% RSLogix 500 project Project - Five_Conveyor_System.RSS, saved by version 8.30.00.16 %
PROJECT "UNTITLED"    % processor: Bul.1763 MicroLogix 1100 Series B %

PROGRAM FILES
  LAD 2 "MAIN"  8 rungs
  LAD 3 "BELT 1"  8 rungs  % Conveyor 1 %
  LAD 4 "BELT 2"  8 rungs  % CONVEYOR 2 %
  LAD 5 "BELT 3"  8 rungs  % CONVEYOR 3 %
  LAD 6 "BELT 4"  8 rungs  % CONVEYOR 4 %
  LAD 7 "BELT 5"  8 rungs  % CONVEYOR 5 %
  LAD 8 "SEQUENCE"  14 rungs  % CONVEYOR OPERATION %

DATA FILES
  O0 OUTPUT  4 elements
  I1 INPUT  6 elements
  S2 STATUS  66 elements
  B3 BINARY  5 elements
  T4 TIMER  25 elements
  C5 COUNTER  5 elements
  R6 CONTROL  1 elements
  N7 INTEGER  5 elements
  F8 FLOAT  1 elements

LADDER 2 "MAIN"
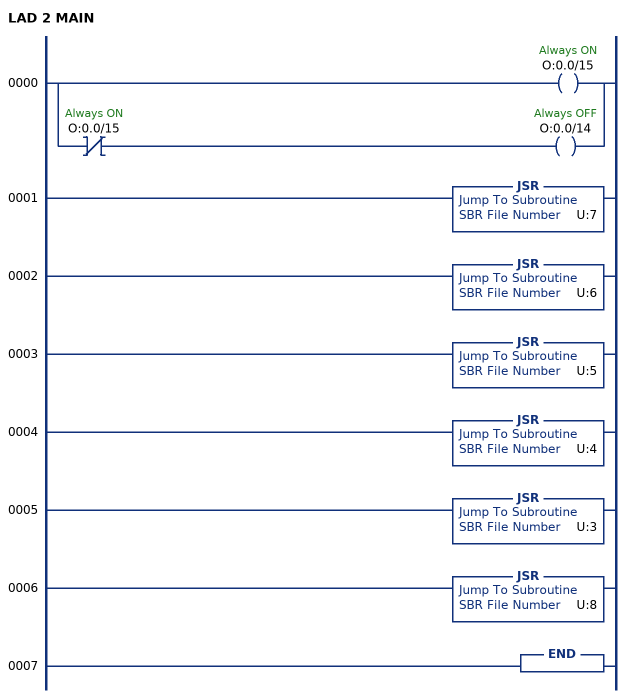
% Rung: 0 %
SOR BST OTE O:0.0/15 NXB XIO O:0.0/15 OTE O:0.0/14 BND EOR
%   O:0.0/15  "Always ON" %
%   O:0.0/14  "Always OFF" %
% Rung: 1 %
SOR JSR U:7 EOR
% Rung: 2 %
SOR JSR U:6 EOR
% Rung: 3 %
SOR JSR U:5 EOR
% Rung: 4 %
SOR JSR U:4 EOR
% Rung: 5 %
SOR JSR U:3 EOR
% Rung: 6 %
SOR JSR U:8 EOR
% Rung: 7 %
SOR END EOR

LADDER 3 "BELT 1"    % Conveyor 1 %
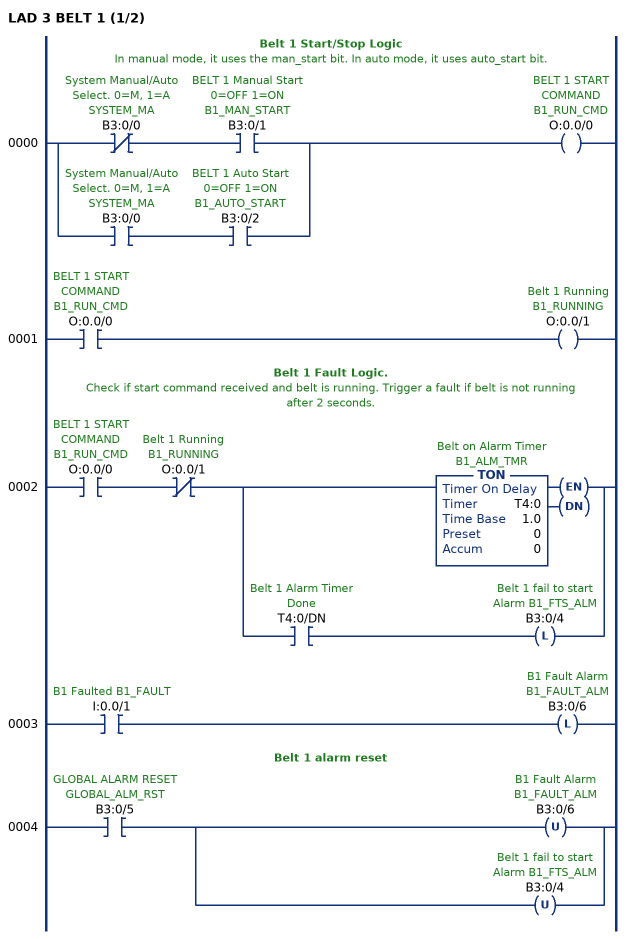
% Rung: 0 %
% TITLE: Belt 1 Start/Stop Logic %
% In manual mode, it uses the man_start bit. In auto mode, it uses auto_start bit. %
SOR BST XIO B3:0/0 XIC B3:0/1 NXB XIC B3:0/0 XIC B3:0/2 BND OTE O:0.0/0 EOR
%   B3:0/0  SYSTEM_MA  "System Manual/Auto Select. 0=M, 1=A" %
%   B3:0/1  B1_MAN_START  "BELT 1 Manual Start 0=OFF 1=ON" %
%   B3:0/2  B1_AUTO_START  "BELT 1 Auto Start 0=OFF 1=ON" %
%   O:0.0/0  B1_RUN_CMD  "BELT 1 START COMMAND" %
% Rung: 1 %
SOR XIC O:0.0/0 OTE O:0.0/1 EOR
%   O:0.0/0  B1_RUN_CMD  "BELT 1 START COMMAND" %
%   O:0.0/1  B1_RUNNING  "Belt 1 Running" %
% Rung: 2 %
% TITLE: Belt 1 Fault Logic. %
% Check if start command received and belt is running. Trigger a fault if belt is not running after 2 seconds. %
SOR XIC O:0.0/0 XIO O:0.0/1 BST TON T4:0 1.0 0 0 NXB XIC T4:0/DN OTL B3:0/4 BND EOR
%   O:0.0/0  B1_RUN_CMD  "BELT 1 START COMMAND" %
%   O:0.0/1  B1_RUNNING  "Belt 1 Running" %
%   T4:0  B1_ALM_TMR  "Belt on Alarm Timer" %
%   T4:0/DN  "Belt 1 Alarm Timer Done" %
%   B3:0/4  B1_FTS_ALM  "Belt 1 fail to start Alarm" %
% Rung: 3 %
SOR XIC I:0.0/1 OTL B3:0/6 EOR
%   I:0.0/1  B1_FAULT  "B1 Faulted" %
%   B3:0/6  B1_FAULT_ALM  "B1 Fault Alarm" %
% Rung: 4 %
% TITLE: Belt 1 alarm reset %
SOR XIC B3:0/5 BST OTU B3:0/6 NXB OTU B3:0/4 BND EOR
%   B3:0/5  GLOBAL_ALM_RST  "GLOBAL ALARM RESET" %
%   B3:0/6  B1_FAULT_ALM  "B1 Fault Alarm" %
%   B3:0/4  B1_FTS_ALM  "Belt 1 fail to start Alarm" %

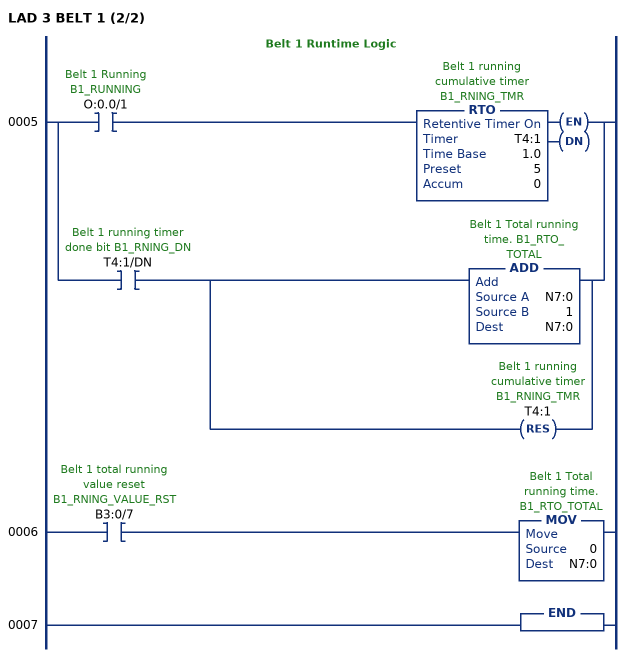
% Rung: 5 %
% TITLE: Belt 1 Runtime Logic %
SOR BST XIC O:0.0/1 RTO T4:1 1.0 5 0 NXB XIC T4:1/DN BST ADD N7:0 1 N7:0 NXB RES T4:1 BND BND EOR
%   O:0.0/1  B1_RUNNING  "Belt 1 Running" %
%   T4:1  B1_RNING_TMR  "Belt 1 running cumulative timer" %
%   T4:1/DN  B1_RNING_DN  "Belt 1 running timer done bit" %
%   N7:0  B1_RTO_TOTAL  "Belt 1 Total running time." %
% Rung: 6 %
SOR XIC B3:0/7 MOV 0 N7:0 EOR
%   B3:0/7  B1_RNING_VALUE_RST  "Belt 1 total running value reset" %
%   N7:0  B1_RTO_TOTAL  "Belt 1 Total running time." %
% Rung: 7 %
SOR END EOR

LADDER 4 "BELT 2"    % CONVEYOR 2 %
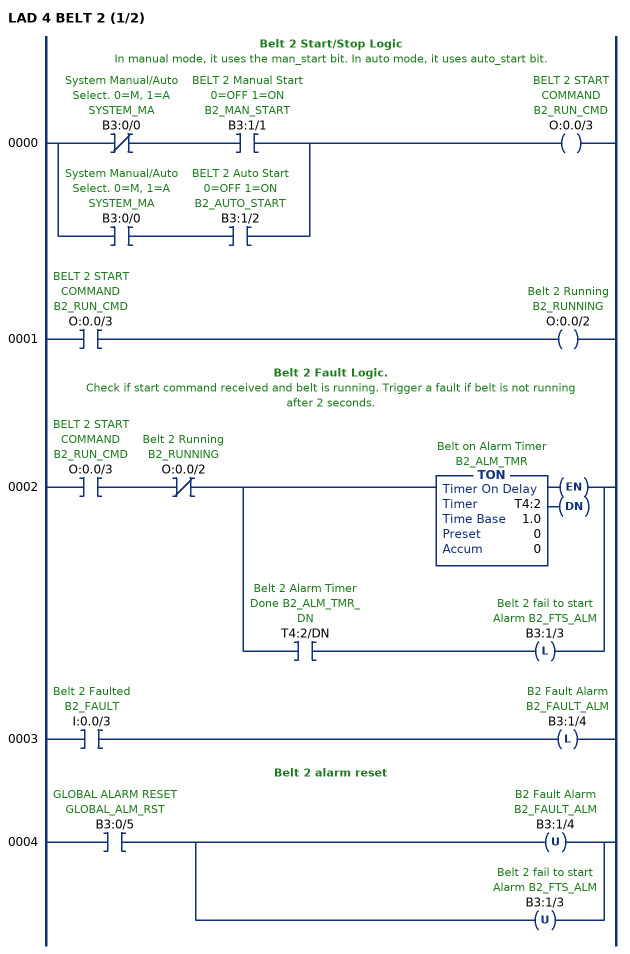
% Rung: 0 %
% TITLE: Belt 2 Start/Stop Logic %
% In manual mode, it uses the man_start bit. In auto mode, it uses auto_start bit. %
SOR BST XIO B3:0/0 XIC B3:1/1 NXB XIC B3:0/0 XIC B3:1/2 BND OTE O:0.0/3 EOR
%   B3:0/0  SYSTEM_MA  "System Manual/Auto Select. 0=M, 1=A" %
%   B3:1/1  B2_MAN_START  "BELT 2 Manual Start 0=OFF 1=ON" %
%   B3:1/2  B2_AUTO_START  "BELT 2 Auto Start 0=OFF 1=ON" %
%   O:0.0/3  B2_RUN_CMD  "BELT 2 START COMMAND" %
% Rung: 1 %
SOR XIC O:0.0/3 OTE O:0.0/2 EOR
%   O:0.0/3  B2_RUN_CMD  "BELT 2 START COMMAND" %
%   O:0.0/2  B2_RUNNING  "Belt 2 Running" %
% Rung: 2 %
% TITLE: Belt 2 Fault Logic. %
% Check if start command received and belt is running. Trigger a fault if belt is not running after 2 seconds. %
SOR XIC O:0.0/3 XIO O:0.0/2 BST TON T4:2 1.0 0 0 NXB XIC T4:2/DN OTL B3:1/3 BND EOR
%   O:0.0/3  B2_RUN_CMD  "BELT 2 START COMMAND" %
%   O:0.0/2  B2_RUNNING  "Belt 2 Running" %
%   T4:2  B2_ALM_TMR  "Belt on Alarm Timer" %
%   T4:2/DN  B2_ALM_TMR_DN  "Belt 2 Alarm Timer Done" %
%   B3:1/3  B2_FTS_ALM  "Belt 2 fail to start Alarm" %
% Rung: 3 %
SOR XIC I:0.0/3 OTL B3:1/4 EOR
%   I:0.0/3  B2_FAULT  "Belt 2 Faulted" %
%   B3:1/4  B2_FAULT_ALM  "B2 Fault Alarm" %
% Rung: 4 %
% TITLE: Belt 2 alarm reset %
SOR XIC B3:0/5 BST OTU B3:1/4 NXB OTU B3:1/3 BND EOR
%   B3:0/5  GLOBAL_ALM_RST  "GLOBAL ALARM RESET" %
%   B3:1/4  B2_FAULT_ALM  "B2 Fault Alarm" %
%   B3:1/3  B2_FTS_ALM  "Belt 2 fail to start Alarm" %

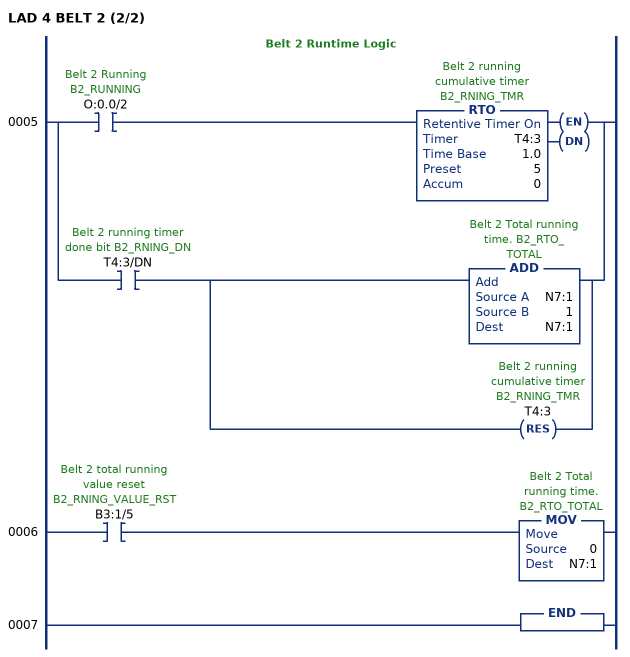
% Rung: 5 %
% TITLE: Belt 2 Runtime Logic %
SOR BST XIC O:0.0/2 RTO T4:3 1.0 5 0 NXB XIC T4:3/DN BST ADD N7:1 1 N7:1 NXB RES T4:3 BND BND EOR
%   O:0.0/2  B2_RUNNING  "Belt 2 Running" %
%   T4:3  B2_RNING_TMR  "Belt 2 running cumulative timer" %
%   T4:3/DN  B2_RNING_DN  "Belt 2 running timer done bit" %
%   N7:1  B2_RTO_TOTAL  "Belt 2 Total running time." %
% Rung: 6 %
SOR XIC B3:1/5 MOV 0 N7:1 EOR
%   B3:1/5  B2_RNING_VALUE_RST  "Belt 2 total running value reset" %
%   N7:1  B2_RTO_TOTAL  "Belt 2 Total running time." %
% Rung: 7 %
SOR END EOR

LADDER 5 "BELT 3"    % CONVEYOR 3 %
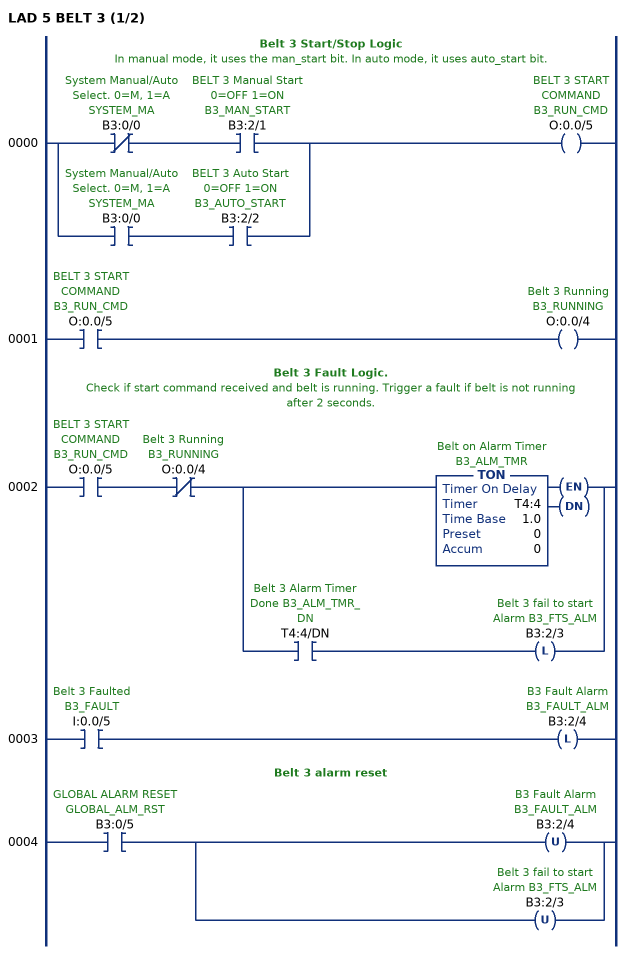
% Rung: 0 %
% TITLE: Belt 3 Start/Stop Logic %
% In manual mode, it uses the man_start bit. In auto mode, it uses auto_start bit. %
SOR BST XIO B3:0/0 XIC B3:2/1 NXB XIC B3:0/0 XIC B3:2/2 BND OTE O:0.0/5 EOR
%   B3:0/0  SYSTEM_MA  "System Manual/Auto Select. 0=M, 1=A" %
%   B3:2/1  B3_MAN_START  "BELT 3 Manual Start 0=OFF 1=ON" %
%   B3:2/2  B3_AUTO_START  "BELT 3 Auto Start 0=OFF 1=ON" %
%   O:0.0/5  B3_RUN_CMD  "BELT 3 START COMMAND" %
% Rung: 1 %
SOR XIC O:0.0/5 OTE O:0.0/4 EOR
%   O:0.0/5  B3_RUN_CMD  "BELT 3 START COMMAND" %
%   O:0.0/4  B3_RUNNING  "Belt 3 Running" %
% Rung: 2 %
% TITLE: Belt 3 Fault Logic. %
% Check if start command received and belt is running. Trigger a fault if belt is not running after 2 seconds. %
SOR XIC O:0.0/5 XIO O:0.0/4 BST TON T4:4 1.0 0 0 NXB XIC T4:4/DN OTL B3:2/3 BND EOR
%   O:0.0/5  B3_RUN_CMD  "BELT 3 START COMMAND" %
%   O:0.0/4  B3_RUNNING  "Belt 3 Running" %
%   T4:4  B3_ALM_TMR  "Belt on Alarm Timer" %
%   T4:4/DN  B3_ALM_TMR_DN  "Belt 3 Alarm Timer Done" %
%   B3:2/3  B3_FTS_ALM  "Belt 3 fail to start Alarm" %
% Rung: 3 %
SOR XIC I:0.0/5 OTL B3:2/4 EOR
%   I:0.0/5  B3_FAULT  "Belt 3 Faulted" %
%   B3:2/4  B3_FAULT_ALM  "B3 Fault Alarm" %
% Rung: 4 %
% TITLE: Belt 3 alarm reset %
SOR XIC B3:0/5 BST OTU B3:2/4 NXB OTU B3:2/3 BND EOR
%   B3:0/5  GLOBAL_ALM_RST  "GLOBAL ALARM RESET" %
%   B3:2/4  B3_FAULT_ALM  "B3 Fault Alarm" %
%   B3:2/3  B3_FTS_ALM  "Belt 3 fail to start Alarm" %

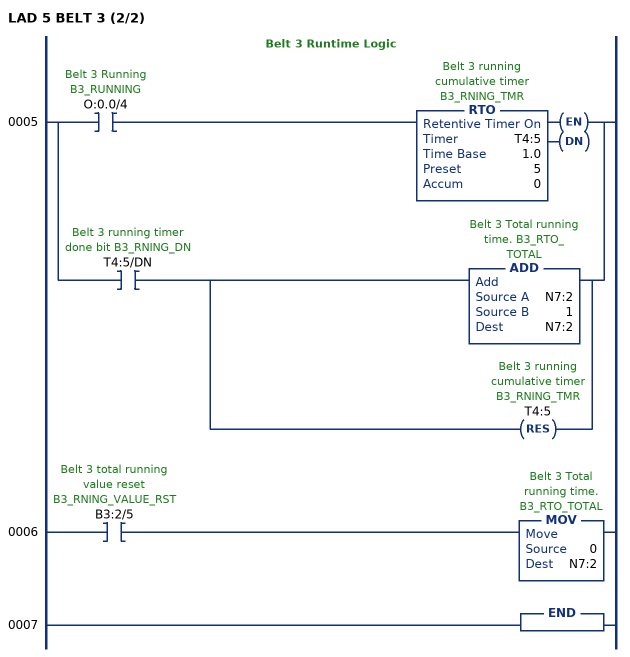
% Rung: 5 %
% TITLE: Belt 3 Runtime Logic %
SOR BST XIC O:0.0/4 RTO T4:5 1.0 5 0 NXB XIC T4:5/DN BST ADD N7:2 1 N7:2 NXB RES T4:5 BND BND EOR
%   O:0.0/4  B3_RUNNING  "Belt 3 Running" %
%   T4:5  B3_RNING_TMR  "Belt 3 running cumulative timer" %
%   T4:5/DN  B3_RNING_DN  "Belt 3 running timer done bit" %
%   N7:2  B3_RTO_TOTAL  "Belt 3 Total running time." %
% Rung: 6 %
SOR XIC B3:2/5 MOV 0 N7:2 EOR
%   B3:2/5  B3_RNING_VALUE_RST  "Belt 3 total running value reset" %
%   N7:2  B3_RTO_TOTAL  "Belt 3 Total running time." %
% Rung: 7 %
SOR END EOR

LADDER 6 "BELT 4"    % CONVEYOR 4 %
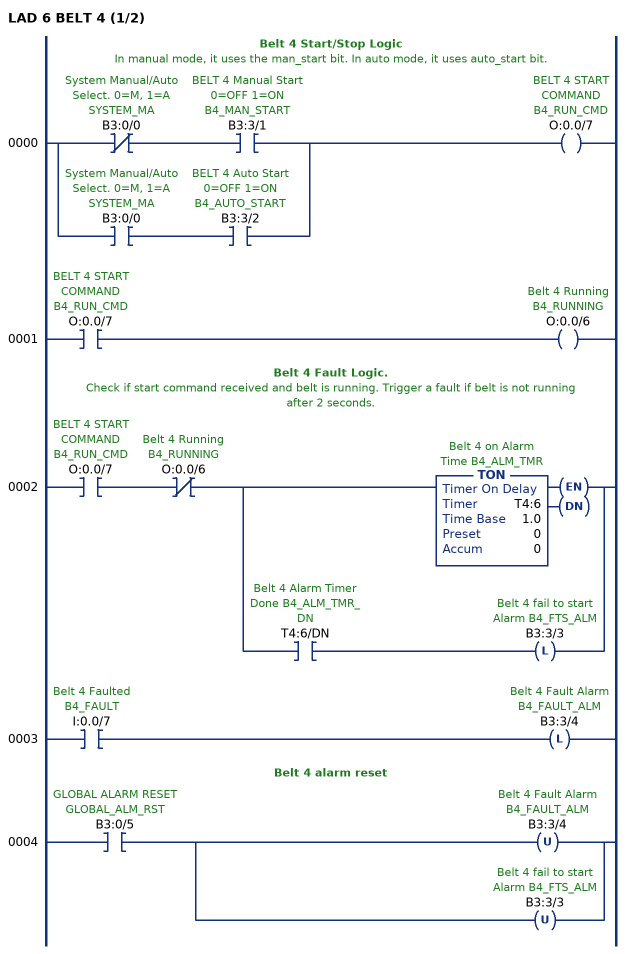
% Rung: 0 %
% TITLE: Belt 4 Start/Stop Logic %
% In manual mode, it uses the man_start bit. In auto mode, it uses auto_start bit. %
SOR BST XIO B3:0/0 XIC B3:3/1 NXB XIC B3:0/0 XIC B3:3/2 BND OTE O:0.0/7 EOR
%   B3:0/0  SYSTEM_MA  "System Manual/Auto Select. 0=M, 1=A" %
%   B3:3/1  B4_MAN_START  "BELT 4 Manual Start 0=OFF 1=ON" %
%   B3:3/2  B4_AUTO_START  "BELT 4 Auto Start 0=OFF 1=ON" %
%   O:0.0/7  B4_RUN_CMD  "BELT 4 START COMMAND" %
% Rung: 1 %
SOR XIC O:0.0/7 OTE O:0.0/6 EOR
%   O:0.0/7  B4_RUN_CMD  "BELT 4 START COMMAND" %
%   O:0.0/6  B4_RUNNING  "Belt 4 Running" %
% Rung: 2 %
% TITLE: Belt 4 Fault Logic. %
% Check if start command received and belt is running. Trigger a fault if belt is not running after 2 seconds. %
SOR XIC O:0.0/7 XIO O:0.0/6 BST TON T4:6 1.0 0 0 NXB XIC T4:6/DN OTL B3:3/3 BND EOR
%   O:0.0/7  B4_RUN_CMD  "BELT 4 START COMMAND" %
%   O:0.0/6  B4_RUNNING  "Belt 4 Running" %
%   T4:6  B4_ALM_TMR  "Belt 4 on Alarm Time" %
%   T4:6/DN  B4_ALM_TMR_DN  "Belt 4 Alarm Timer Done" %
%   B3:3/3  B4_FTS_ALM  "Belt 4 fail to start Alarm" %
% Rung: 3 %
SOR XIC I:0.0/7 OTL B3:3/4 EOR
%   I:0.0/7  B4_FAULT  "Belt 4 Faulted" %
%   B3:3/4  B4_FAULT_ALM  "Belt 4 Fault Alarm" %
% Rung: 4 %
% TITLE: Belt 4 alarm reset %
SOR XIC B3:0/5 BST OTU B3:3/4 NXB OTU B3:3/3 BND EOR
%   B3:0/5  GLOBAL_ALM_RST  "GLOBAL ALARM RESET" %
%   B3:3/4  B4_FAULT_ALM  "Belt 4 Fault Alarm" %
%   B3:3/3  B4_FTS_ALM  "Belt 4 fail to start Alarm" %

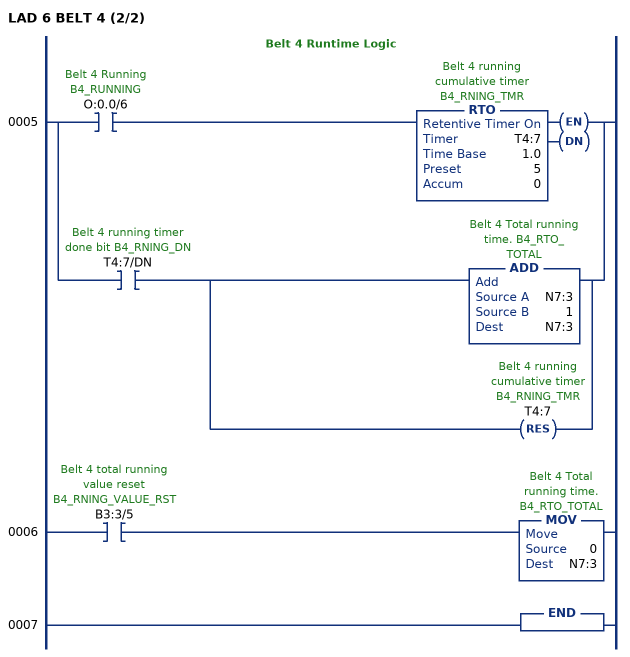
% Rung: 5 %
% TITLE: Belt 4 Runtime Logic %
SOR BST XIC O:0.0/6 RTO T4:7 1.0 5 0 NXB XIC T4:7/DN BST ADD N7:3 1 N7:3 NXB RES T4:7 BND BND EOR
%   O:0.0/6  B4_RUNNING  "Belt 4 Running" %
%   T4:7  B4_RNING_TMR  "Belt 4 running cumulative timer" %
%   T4:7/DN  B4_RNING_DN  "Belt 4 running timer done bit" %
%   N7:3  B4_RTO_TOTAL  "Belt 4 Total running time." %
% Rung: 6 %
SOR XIC B3:3/5 MOV 0 N7:3 EOR
%   B3:3/5  B4_RNING_VALUE_RST  "Belt 4 total running value reset" %
%   N7:3  B4_RTO_TOTAL  "Belt 4 Total running time." %
% Rung: 7 %
SOR END EOR

LADDER 7 "BELT 5"    % CONVEYOR 5 %
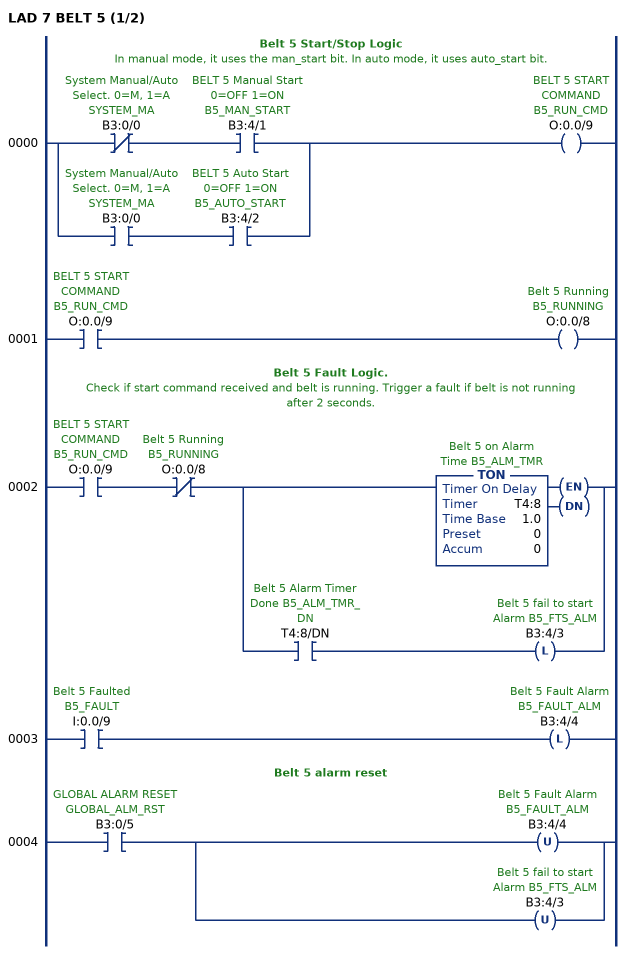
% Rung: 0 %
% TITLE: Belt 5 Start/Stop Logic %
% In manual mode, it uses the man_start bit. In auto mode, it uses auto_start bit. %
SOR BST XIO B3:0/0 XIC B3:4/1 NXB XIC B3:0/0 XIC B3:4/2 BND OTE O:0.0/9 EOR
%   B3:0/0  SYSTEM_MA  "System Manual/Auto Select. 0=M, 1=A" %
%   B3:4/1  B5_MAN_START  "BELT 5 Manual Start 0=OFF 1=ON" %
%   B3:4/2  B5_AUTO_START  "BELT 5 Auto Start 0=OFF 1=ON" %
%   O:0.0/9  B5_RUN_CMD  "BELT 5 START COMMAND" %
% Rung: 1 %
SOR XIC O:0.0/9 OTE O:0.0/8 EOR
%   O:0.0/9  B5_RUN_CMD  "BELT 5 START COMMAND" %
%   O:0.0/8  B5_RUNNING  "Belt 5 Running" %
% Rung: 2 %
% TITLE: Belt 5 Fault Logic. %
% Check if start command received and belt is running. Trigger a fault if belt is not running after 2 seconds. %
SOR XIC O:0.0/9 XIO O:0.0/8 BST TON T4:8 1.0 0 0 NXB XIC T4:8/DN OTL B3:4/3 BND EOR
%   O:0.0/9  B5_RUN_CMD  "BELT 5 START COMMAND" %
%   O:0.0/8  B5_RUNNING  "Belt 5 Running" %
%   T4:8  B5_ALM_TMR  "Belt 5 on Alarm Time" %
%   T4:8/DN  B5_ALM_TMR_DN  "Belt 5 Alarm Timer Done" %
%   B3:4/3  B5_FTS_ALM  "Belt 5 fail to start Alarm" %
% Rung: 3 %
SOR XIC I:0.0/9 OTL B3:4/4 EOR
%   I:0.0/9  B5_FAULT  "Belt 5 Faulted" %
%   B3:4/4  B5_FAULT_ALM  "Belt 5 Fault Alarm" %
% Rung: 4 %
% TITLE: Belt 5 alarm reset %
SOR XIC B3:0/5 BST OTU B3:4/4 NXB OTU B3:4/3 BND EOR
%   B3:0/5  GLOBAL_ALM_RST  "GLOBAL ALARM RESET" %
%   B3:4/4  B5_FAULT_ALM  "Belt 5 Fault Alarm" %
%   B3:4/3  B5_FTS_ALM  "Belt 5 fail to start Alarm" %

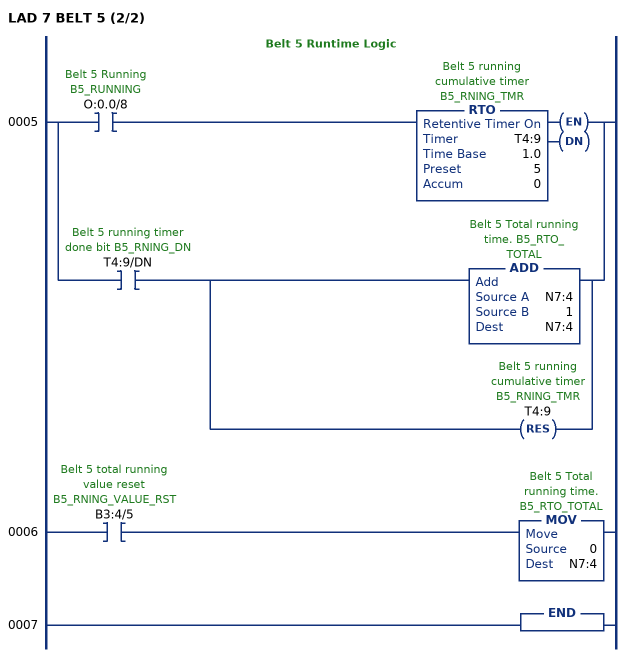
% Rung: 5 %
% TITLE: Belt 5 Runtime Logic %
SOR BST XIC O:0.0/8 RTO T4:9 1.0 5 0 NXB XIC T4:9/DN BST ADD N7:4 1 N7:4 NXB RES T4:9 BND BND EOR
%   O:0.0/8  B5_RUNNING  "Belt 5 Running" %
%   T4:9  B5_RNING_TMR  "Belt 5 running cumulative timer" %
%   T4:9/DN  B5_RNING_DN  "Belt 5 running timer done bit" %
%   N7:4  B5_RTO_TOTAL  "Belt 5 Total running time." %
% Rung: 6 %
SOR XIC B3:4/5 MOV 0 N7:4 EOR
%   B3:4/5  B5_RNING_VALUE_RST  "Belt 5 total running value reset" %
%   N7:4  B5_RTO_TOTAL  "Belt 5 Total running time." %
% Rung: 7 %
SOR END EOR

LADDER 8 "SEQUENCE"    % CONVEYOR OPERATION %
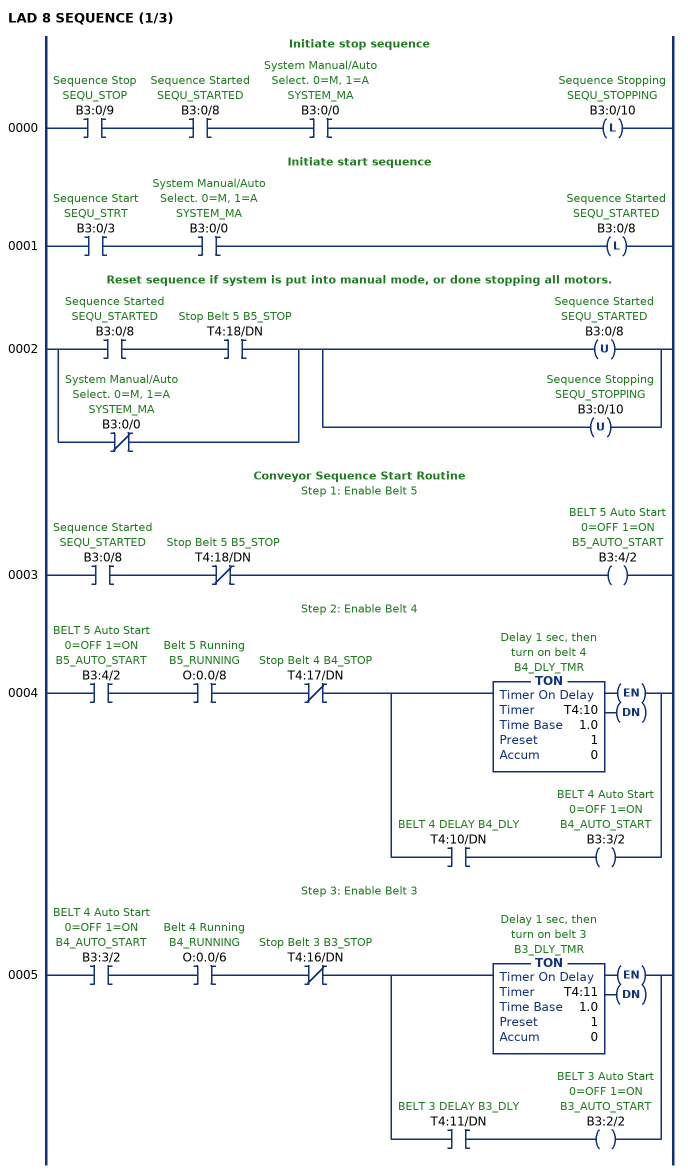
% Rung: 0 %
% TITLE: Initiate stop sequence %
SOR XIC B3:0/9 XIC B3:0/8 XIC B3:0/0 OTL B3:0/10 EOR
%   B3:0/9  SEQU_STOP  "Sequence Stop" %
%   B3:0/8  SEQU_STARTED  "Sequence Started" %
%   B3:0/0  SYSTEM_MA  "System Manual/Auto Select. 0=M, 1=A" %
%   B3:0/10  SEQU_STOPPING  "Sequence Stopping" %
% Rung: 1 %
% TITLE: Initiate start sequence %
SOR XIC B3:0/3 XIC B3:0/0 OTL B3:0/8 EOR
%   B3:0/3  SEQU_STRT  "Sequence Start" %
%   B3:0/0  SYSTEM_MA  "System Manual/Auto Select. 0=M, 1=A" %
%   B3:0/8  SEQU_STARTED  "Sequence Started" %
% Rung: 2 %
% TITLE: Reset sequence if system is put into manual mode, or done stopping all motors. %
SOR BST XIC B3:0/8 XIC T4:18/DN NXB XIO B3:0/0 BND BST OTU B3:0/8 NXB OTU B3:0/10 BND EOR
%   B3:0/8  SEQU_STARTED  "Sequence Started" %
%   T4:18/DN  B5_STOP  "Stop Belt 5" %
%   B3:0/0  SYSTEM_MA  "System Manual/Auto Select. 0=M, 1=A" %
%   B3:0/10  SEQU_STOPPING  "Sequence Stopping" %
% Rung: 3 %
% TITLE: Conveyor Sequence Start Routine %
% Step 1: Enable Belt 5 %
SOR XIC B3:0/8 XIO T4:18/DN OTE B3:4/2 EOR
%   B3:0/8  SEQU_STARTED  "Sequence Started" %
%   T4:18/DN  B5_STOP  "Stop Belt 5" %
%   B3:4/2  B5_AUTO_START  "BELT 5 Auto Start 0=OFF 1=ON" %
% Rung: 4 %
% Step 2: Enable Belt 4 %
SOR XIC B3:4/2 XIC O:0.0/8 XIO T4:17/DN BST TON T4:10 1.0 1 0 NXB XIC T4:10/DN OTE B3:3/2 BND EOR
%   B3:4/2  B5_AUTO_START  "BELT 5 Auto Start 0=OFF 1=ON" %
%   O:0.0/8  B5_RUNNING  "Belt 5 Running" %
%   T4:17/DN  B4_STOP  "Stop Belt 4" %
%   T4:10  B4_DLY_TMR  "Delay 1 sec, then turn on belt 4" %
%   T4:10/DN  B4_DLY  "BELT 4 DELAY" %
%   B3:3/2  B4_AUTO_START  "BELT 4 Auto Start 0=OFF 1=ON" %
% Rung: 5 %
% Step 3: Enable Belt 3 %
SOR XIC B3:3/2 XIC O:0.0/6 XIO T4:16/DN BST TON T4:11 1.0 1 0 NXB XIC T4:11/DN OTE B3:2/2 BND EOR
%   B3:3/2  B4_AUTO_START  "BELT 4 Auto Start 0=OFF 1=ON" %
%   O:0.0/6  B4_RUNNING  "Belt 4 Running" %
%   T4:16/DN  B3_STOP  "Stop Belt 3" %
%   T4:11  B3_DLY_TMR  "Delay 1 sec, then turn on belt 3" %
%   T4:11/DN  B3_DLY  "BELT 3 DELAY" %
%   B3:2/2  B3_AUTO_START  "BELT 3 Auto Start 0=OFF 1=ON" %

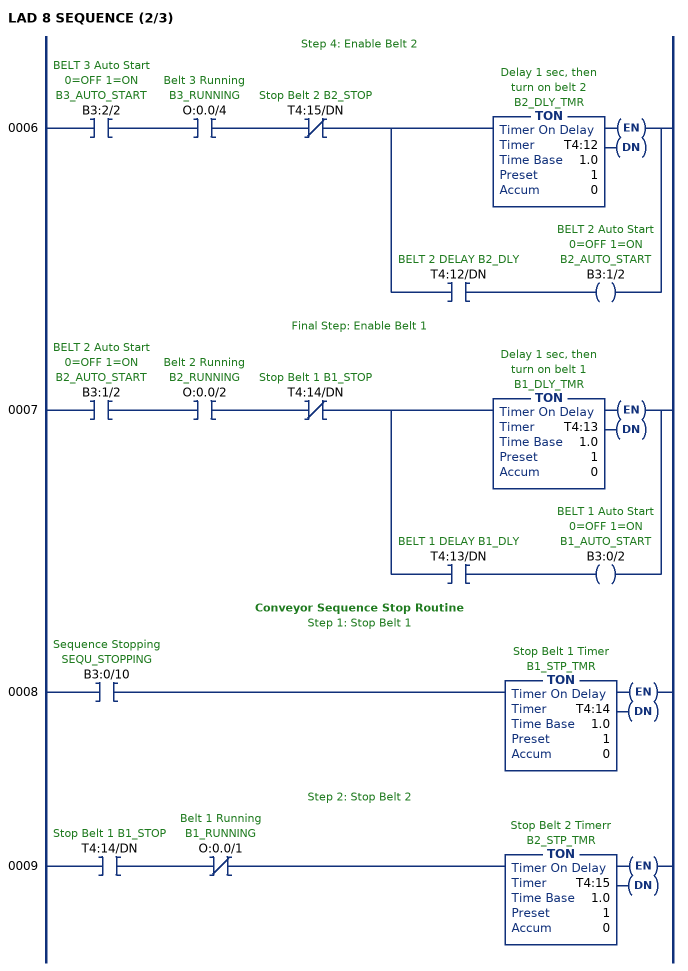
% Rung: 6 %
% Step 4: Enable Belt 2 %
SOR XIC B3:2/2 XIC O:0.0/4 XIO T4:15/DN BST TON T4:12 1.0 1 0 NXB XIC T4:12/DN OTE B3:1/2 BND EOR
%   B3:2/2  B3_AUTO_START  "BELT 3 Auto Start 0=OFF 1=ON" %
%   O:0.0/4  B3_RUNNING  "Belt 3 Running" %
%   T4:15/DN  B2_STOP  "Stop Belt 2" %
%   T4:12  B2_DLY_TMR  "Delay 1 sec, then turn on belt 2" %
%   T4:12/DN  B2_DLY  "BELT 2 DELAY" %
%   B3:1/2  B2_AUTO_START  "BELT 2 Auto Start 0=OFF 1=ON" %
% Rung: 7 %
% Final Step: Enable Belt 1 %
SOR XIC B3:1/2 XIC O:0.0/2 XIO T4:14/DN BST TON T4:13 1.0 1 0 NXB XIC T4:13/DN OTE B3:0/2 BND EOR
%   B3:1/2  B2_AUTO_START  "BELT 2 Auto Start 0=OFF 1=ON" %
%   O:0.0/2  B2_RUNNING  "Belt 2 Running" %
%   T4:14/DN  B1_STOP  "Stop Belt 1" %
%   T4:13  B1_DLY_TMR  "Delay 1 sec, then turn on belt 1" %
%   T4:13/DN  B1_DLY  "BELT 1 DELAY" %
%   B3:0/2  B1_AUTO_START  "BELT 1 Auto Start 0=OFF 1=ON" %
% Rung: 8 %
% TITLE: Conveyor Sequence Stop Routine %
% Step 1: Stop Belt 1 %
SOR XIC B3:0/10 TON T4:14 1.0 1 0 EOR
%   B3:0/10  SEQU_STOPPING  "Sequence Stopping" %
%   T4:14  B1_STP_TMR  "Stop Belt 1 Timer" %
% Rung: 9 %
% Step 2: Stop Belt 2 %
SOR XIC T4:14/DN XIO O:0.0/1 TON T4:15 1.0 1 0 EOR
%   T4:14/DN  B1_STOP  "Stop Belt 1" %
%   O:0.0/1  B1_RUNNING  "Belt 1 Running" %
%   T4:15  B2_STP_TMR  "Stop Belt 2 Timerr" %

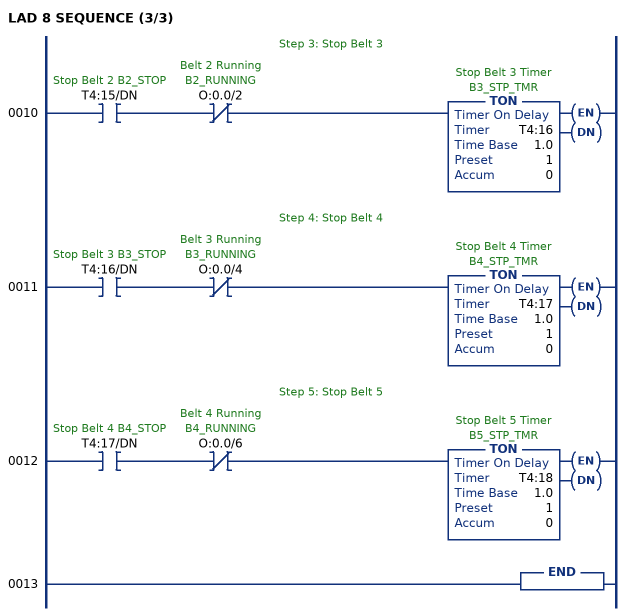
% Rung: 10 %
% Step 3: Stop Belt 3 %
SOR XIC T4:15/DN XIO O:0.0/2 TON T4:16 1.0 1 0 EOR
%   T4:15/DN  B2_STOP  "Stop Belt 2" %
%   O:0.0/2  B2_RUNNING  "Belt 2 Running" %
%   T4:16  B3_STP_TMR  "Stop Belt 3 Timer" %
% Rung: 11 %
% Step 4: Stop Belt 4 %
SOR XIC T4:16/DN XIO O:0.0/4 TON T4:17 1.0 1 0 EOR
%   T4:16/DN  B3_STOP  "Stop Belt 3" %
%   O:0.0/4  B3_RUNNING  "Belt 3 Running" %
%   T4:17  B4_STP_TMR  "Stop Belt 4 Timer" %
% Rung: 12 %
% Step 5: Stop Belt 5 %
SOR XIC T4:17/DN XIO O:0.0/6 TON T4:18 1.0 1 0 EOR
%   T4:17/DN  B4_STOP  "Stop Belt 4" %
%   O:0.0/6  B4_RUNNING  "Belt 4 Running" %
%   T4:18  B5_STP_TMR  "Stop Belt 5 Timer" %
% Rung: 13 %
SOR END EOR

OTHER DOCUMENTED ADDRESSES
  C5:0  B1_RNING_CNTR  "Belt 1 running counter"
  C5:1  B2_RNING_CNTR  "Belt 2 running counter"
  C5:2  B3_RNING_CNTR  "Belt 3 running counter"
  C5:3  B4_RNING_CNTR  "Belt 4 running counter"
  C5:4  B5_RNING_CNTR  "Belt 5 running counter"
  DFILE:0  "OUTPUT"
  DFILE:1  "INPUT"
  DFILE:2  "STATUS"
  DFILE:3  "BINARY"
  DFILE:4  "TIMER"
  DFILE:5  "COUNTER"
  DFILE:6  "CONTROL"
  DFILE:7  "INTEGER"
  DFILE:8  "FLOAT"
  I:1.0/0  "Manual Stop"
  I:1.0/2  BELT1_STOP  "Manual Stop"

COMMENTS NOT ATTACHED TO A CURRENT RUNG
  O:0.0/0: Belt 1 Start/Stop Logic / In manual mode, it uses the man_start bit. In auto mode, it uses auto_start bit.
  B3:3/2: Step 2: Enable Belt 4
  B3:2/2: Step 3: Enable Belt 3

DATA TABLE (non-zero values as saved)
DATA T4
% .PRE .ACC %
% T4:1 % 5 0
% T4:3 % 5 0
% T4:5 % 5 0
% T4:7 % 5 0
% T4:9 % 5 0
% T4:10 % 1 0
% T4:11 % 1 0
% T4:12 % 1 0
% T4:13 % 1 0
% T4:14 % 1 0
% T4:15 % 1 0
% T4:16 % 1 0
% T4:17 % 1 0
% T4:18 % 1 0
